PROGRAM Axis05_Rotation_1
VAR
	Axis05: AXIS_REF;											//회전축
	Axis05_MC_Home: FB_HomeBeforeMoveAX8000;
	Axis05_MC_Power: MC_Power;
	Axis05_Status: MC_ReadStatus;
	Axis05_Position_Read: MC_ReadActualPosition;
	Axis05_Velocity_Read: MC_ReadActualVelocity;
	Axis05_Reset: MC_Reset;										//모터 알람 리셋
	Axis05_Stop: MC_Stop;										//모터 정지
	Axis05_Press_Move: MC_MoveAbsolute;
	Axis05_Home_Pos_Move: MC_MoveAbsolute;
	Axis05_Wait_Pos_Move: MC_MoveAbsolute;
	Axis05_Target_Pos_Move: MC_MoveAbsolute;
	Axis05_Work_End_Move: MC_MoveAbsolute;
	Axis05_Jog: MC_Jog;
	
	Always_ON	:	BOOL	:=TRUE	;//상시 ON
	Always_OFF	:	BOOL	:=FALSE	;//상시 OFF

	Home_Interlock			:	BOOL	;
	Home_Pos_Interlock		: 	BOOL	;
	Wait_Pos_Interlock		:	BOOL	;
	Target_Pos_Interlock	:	BOOL	;
	Work_End_POs_Interlock	:	BOOL	;
	Axis05_Calibration: MC_MoveAbsolute;
END_VAR
VAR // added by the converter: edge detectors and wires of the graphical bodies
    _rt1, _rt2, _rt3, _rt4, _rt5, _rt6 : R_TRIG;
    _w1, _w2 : BOOL;
END_VAR

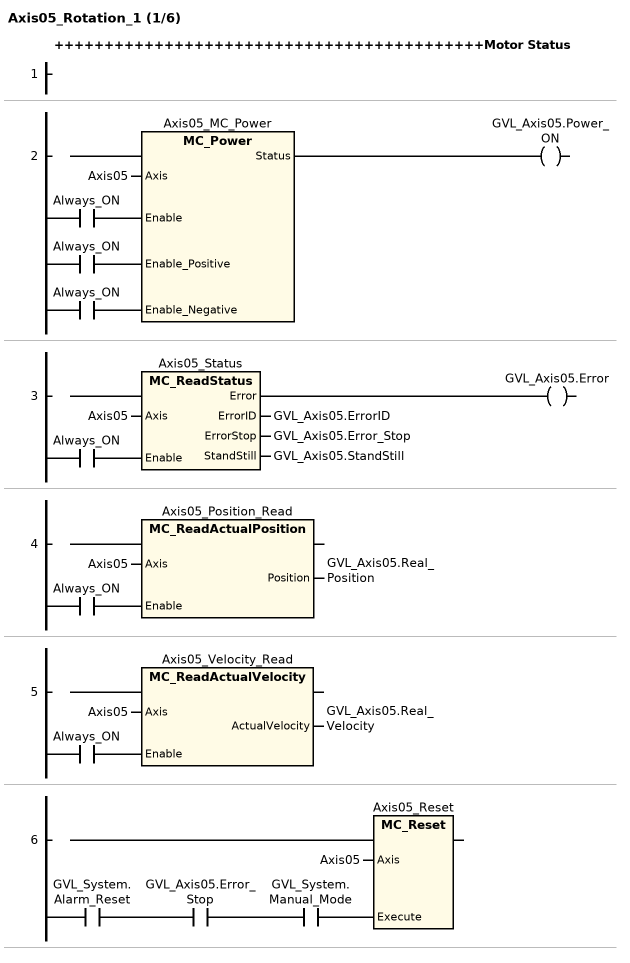
// NETWORK 1: +++++++++++++++++++++++++++++++++++++++++++Motor Status

// NETWORK 2
Axis05_MC_Power(
    Axis := Axis05,
    Enable := Always_ON,
    Enable_Positive := Always_ON,
    Enable_Negative := Always_ON); // MC_Power
GVL_Axis05.Power_ON := Axis05_MC_Power.Status;

// NETWORK 3
Axis05_Status(
    Axis := Axis05,
    Enable := Always_ON,
    Error => GVL_Axis05.Error,
    ErrorID => GVL_Axis05.ErrorID,
    ErrorStop => GVL_Axis05.Error_Stop,
    StandStill => GVL_Axis05.StandStill); // MC_ReadStatus

// NETWORK 4
Axis05_Position_Read(Axis := Axis05, Enable := Always_ON, Position => GVL_Axis05.Real_Position); // MC_ReadActualPosition

// NETWORK 5
Axis05_Velocity_Read(Axis := Axis05, Enable := Always_ON, ActualVelocity => GVL_Axis05.Real_Velocity); // MC_ReadActualVelocity

// NETWORK 6
Axis05_Reset(Axis := Axis05, Execute := GVL_System.Alarm_Reset AND GVL_Axis05.Error_Stop AND GVL_System.Manual_Mode); // MC_Reset

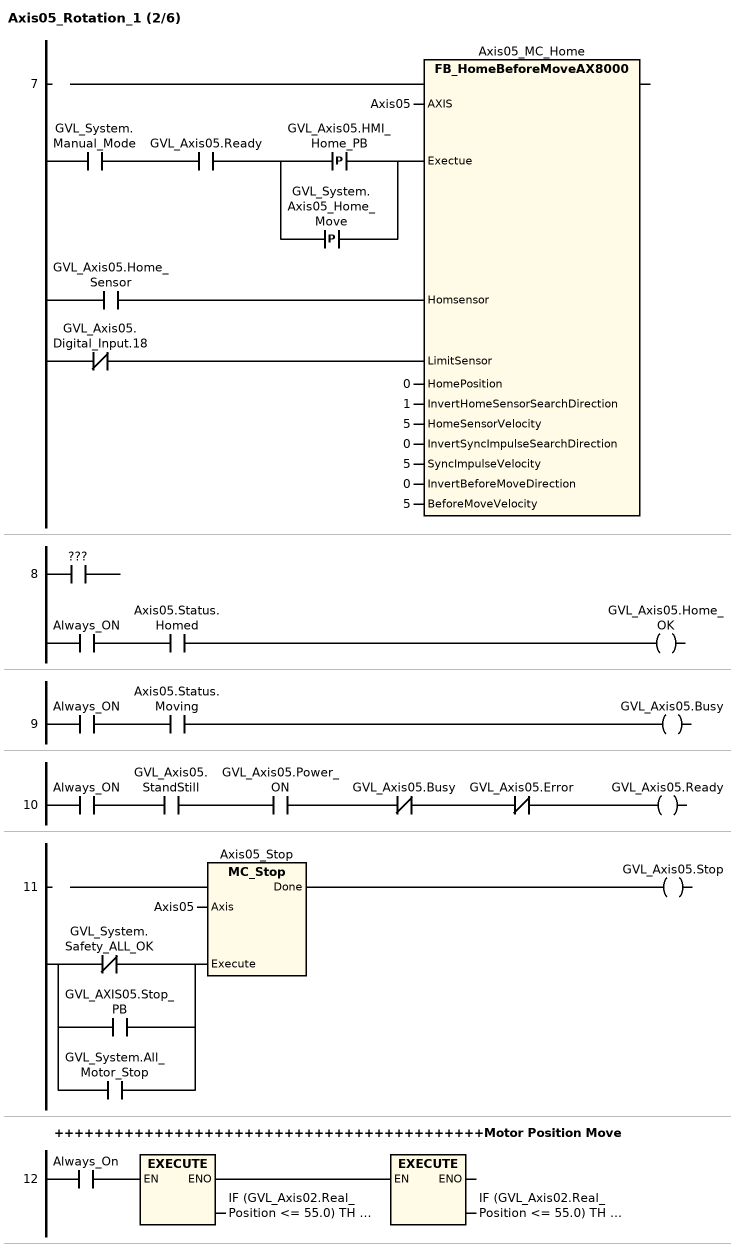
// NETWORK 7
_rt1(CLK := GVL_Axis05.HMI_Home_PB);
_rt2(CLK := GVL_System.Axis05_Home_Move);
Axis05_MC_Home(
    AXIS := Axis05,
    Exectue := GVL_System.Manual_Mode AND GVL_Axis05.Ready AND (_rt1.Q OR _rt2.Q),
    Homsensor := GVL_Axis05.Home_Sensor,
    LimitSensor := NOT GVL_Axis05.Digital_Input.18,
    HomePosition := 0,
    InvertHomeSensorSearchDirection := 1,
    HomeSensorVelocity := 5,
    InvertSyncImpulseSearchDirection := 0,
    SyncImpulseVelocity := 5,
    InvertBeforeMoveDirection := 0,
    BeforeMoveVelocity := 5); // FB_HomeBeforeMoveAX8000

// NETWORK 8
GVL_Axis05.Home_OK := Always_ON AND Axis05.Status.Homed;

// NETWORK 9
GVL_Axis05.Busy := Always_ON AND Axis05.Status.Moving;

// NETWORK 10
GVL_Axis05.Ready := Always_ON AND GVL_Axis05.StandStill AND GVL_Axis05.Power_ON AND NOT GVL_Axis05.Busy AND NOT GVL_Axis05.Error;

// NETWORK 11
Axis05_Stop(Axis := Axis05, Execute := NOT GVL_System.Safety_ALL_OK OR GVL_AXIS05.Stop_PB OR GVL_System.All_Motor_Stop); // MC_Stop
GVL_Axis05.Stop := Axis05_Stop.Done;

// NETWORK 12: +++++++++++++++++++++++++++++++++++++++++++Motor Position Move
_w1 := Always_On;
IF _w1 THEN
    IF (GVL_Axis02.Real_Position <= 55.0) THEN
        Home_Pos_Interlock := TRUE;
    ELSE
        IF (GVL_Axis05.Home_Position_Data >= -1.5) AND 
           (GVL_Axis05.Home_Position_Data <= 2.5) THEN
            Home_Pos_Interlock := TRUE;
        ELSE 
           Home_Pos_Interlock := FALSE;
        END_IF;
    END_IF;
END_IF
IF _w1 THEN
    IF (GVL_Axis02.Real_Position <= 55.0) THEN
        Wait_Pos_Interlock := TRUE;
    ELSE
        IF (GVL_Axis05.Wait_Position_Data >= -1.5) AND 
           (GVL_Axis05.Wait_Position_Data <= 2.5) THEN
            Wait_Pos_Interlock := TRUE;
        ELSE 
           Wait_Pos_Interlock := FALSE;
        END_IF;
    END_IF;
END_IF

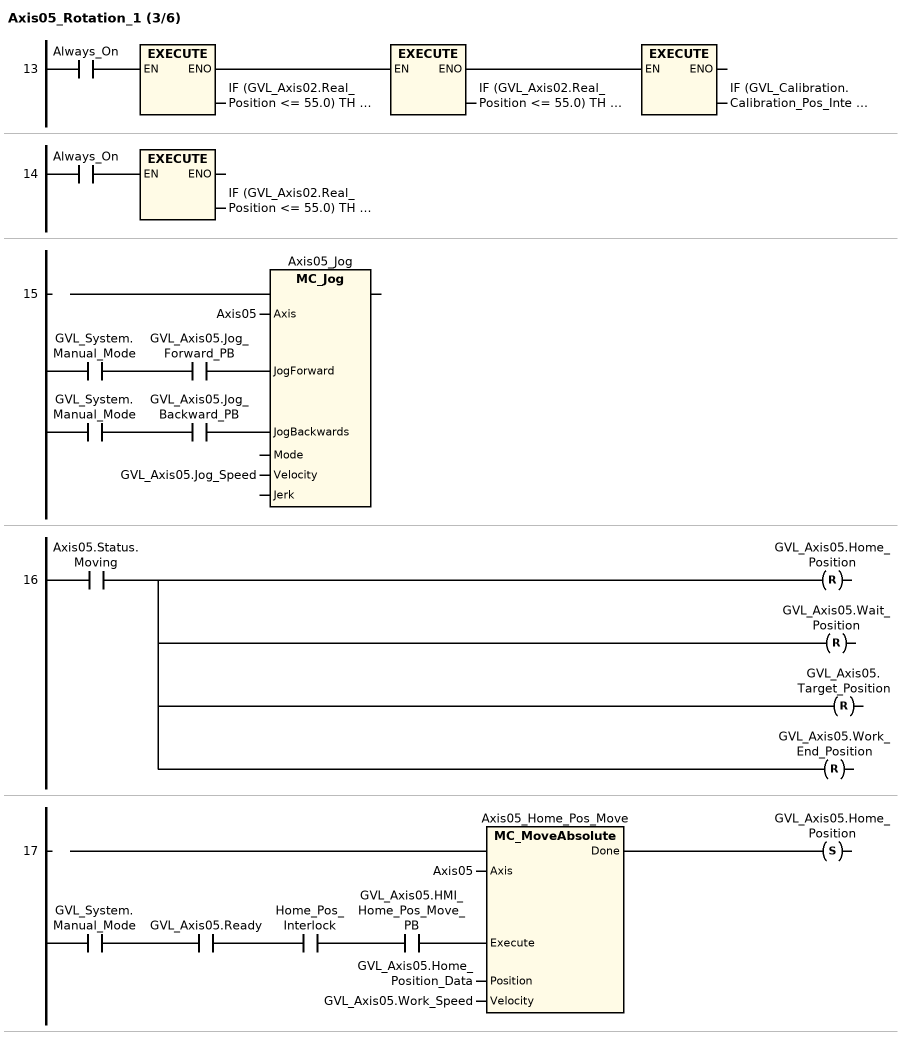
// NETWORK 13
_w2 := Always_On;
IF _w2 THEN
    IF (GVL_Axis02.Real_Position <= 55.0) THEN
        Target_Pos_Interlock := TRUE;
    ELSE
        IF (GVL_Axis05.Target_Position_Data >= -1.5) AND 
           (GVL_Axis05.Target_Position_Data <= 2.5) THEN
            Target_Pos_Interlock := TRUE;
        ELSE 
           Target_Pos_Interlock := FALSE;
        END_IF;
    END_IF;
END_IF
IF _w2 THEN
    IF (GVL_Axis02.Real_Position <= 55.0) THEN
        Work_End_Pos_Interlock := TRUE;
    ELSE
        IF (GVL_Axis05.Work_End_Position_Data >= -1.5) AND 
           (GVL_Axis05.Work_End_Position_Data <= 2.5) THEN
            Work_End_Pos_Interlock := TRUE;
        ELSE 
           Work_End_Pos_Interlock := FALSE;
        END_IF;
    END_IF;
END_IF
IF _w2 THEN
    IF (GVL_Calibration.Calibration_Pos_Interlock = TRUE) AND (Home_Pos_Interlock = TRUE)
    AND (Wait_Pos_Interlock = TRUE) AND (Target_Pos_Interlock = TRUE) AND (Work_End_POs_Interlock = TRUE) THEN
    	GVL_Axis05.Interlock := TRUE;
    	ELSE
    	GVL_Axis05.Interlock := FALSE;	
    
    END_IF
END_IF

// NETWORK 14
IF Always_On THEN
    IF (GVL_Axis02.Real_Position <= 55.0) THEN
        Home_Interlock := TRUE;
    ELSE
           Home_Interlock := FALSE;
    END_IF;
END_IF

// NETWORK 15
Axis05_Jog(
    Axis := Axis05,
    JogForward := GVL_System.Manual_Mode AND GVL_Axis05.Jog_Forward_PB,
    JogBackwards := GVL_System.Manual_Mode AND GVL_Axis05.Jog_Backward_PB,
    Velocity := GVL_Axis05.Jog_Speed); // MC_Jog

// NETWORK 16
GVL_Axis05.Home_Position R= Axis05.Status.Moving;
GVL_Axis05.Wait_Position R= Axis05.Status.Moving;
GVL_Axis05.Target_Position R= Axis05.Status.Moving;
GVL_Axis05.Work_End_Position R= Axis05.Status.Moving;

// NETWORK 17
Axis05_Home_Pos_Move(
    Axis := Axis05,
    Execute := GVL_System.Manual_Mode AND GVL_Axis05.Ready AND Home_Pos_Interlock AND GVL_Axis05.HMI_Home_Pos_Move_PB,
    Position := GVL_Axis05.Home_Position_Data,
    Velocity := GVL_Axis05.Work_Speed); // MC_MoveAbsolute
GVL_Axis05.Home_Position S= Axis05_Home_Pos_Move.Done;

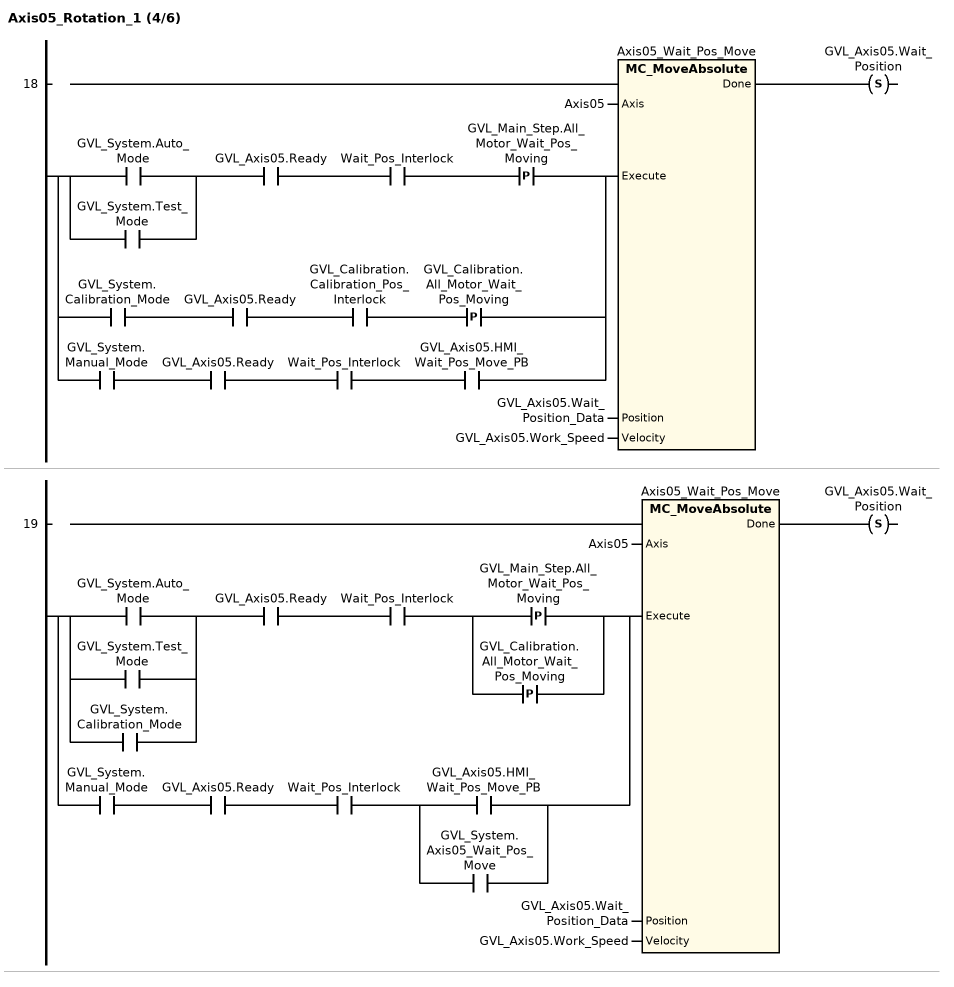
// NETWORK 18
_rt3(CLK := GVL_Main_Step.All_Motor_Wait_Pos_Moving);
_rt4(CLK := GVL_Calibration.All_Motor_Wait_Pos_Moving);
Axis05_Wait_Pos_Move(
    Axis := Axis05,
    Execute := (GVL_System.Auto_Mode OR GVL_System.Test_Mode) AND GVL_Axis05.Ready AND Wait_Pos_Interlock AND _rt3.Q OR GVL_System.Calibration_Mode AND GVL_Axis05.Ready AND GVL_Calibration.Calibration_Pos_Interlock AND _rt4.Q OR GVL_System.Manual_Mode AND GVL_Axis05.Ready AND Wait_Pos_Interlock AND GVL_Axis05.HMI_Wait_Pos_Move_PB,
    Position := GVL_Axis05.Wait_Position_Data,
    Velocity := GVL_Axis05.Work_Speed); // MC_MoveAbsolute
GVL_Axis05.Wait_Position S= Axis05_Wait_Pos_Move.Done;

// NETWORK 19
_rt5(CLK := GVL_Main_Step.All_Motor_Wait_Pos_Moving);
_rt6(CLK := GVL_Calibration.All_Motor_Wait_Pos_Moving);
Axis05_Wait_Pos_Move(
    Axis := Axis05,
    Execute := (GVL_System.Auto_Mode OR GVL_System.Test_Mode OR GVL_System.Calibration_Mode) AND GVL_Axis05.Ready AND Wait_Pos_Interlock AND (_rt5.Q OR _rt6.Q) OR GVL_System.Manual_Mode AND GVL_Axis05.Ready AND Wait_Pos_Interlock AND (GVL_Axis05.HMI_Wait_Pos_Move_PB OR GVL_System.Axis05_Wait_Pos_Move),
    Position := GVL_Axis05.Wait_Position_Data,
    Velocity := GVL_Axis05.Work_Speed); // MC_MoveAbsolute
GVL_Axis05.Wait_Position S= Axis05_Wait_Pos_Move.Done;

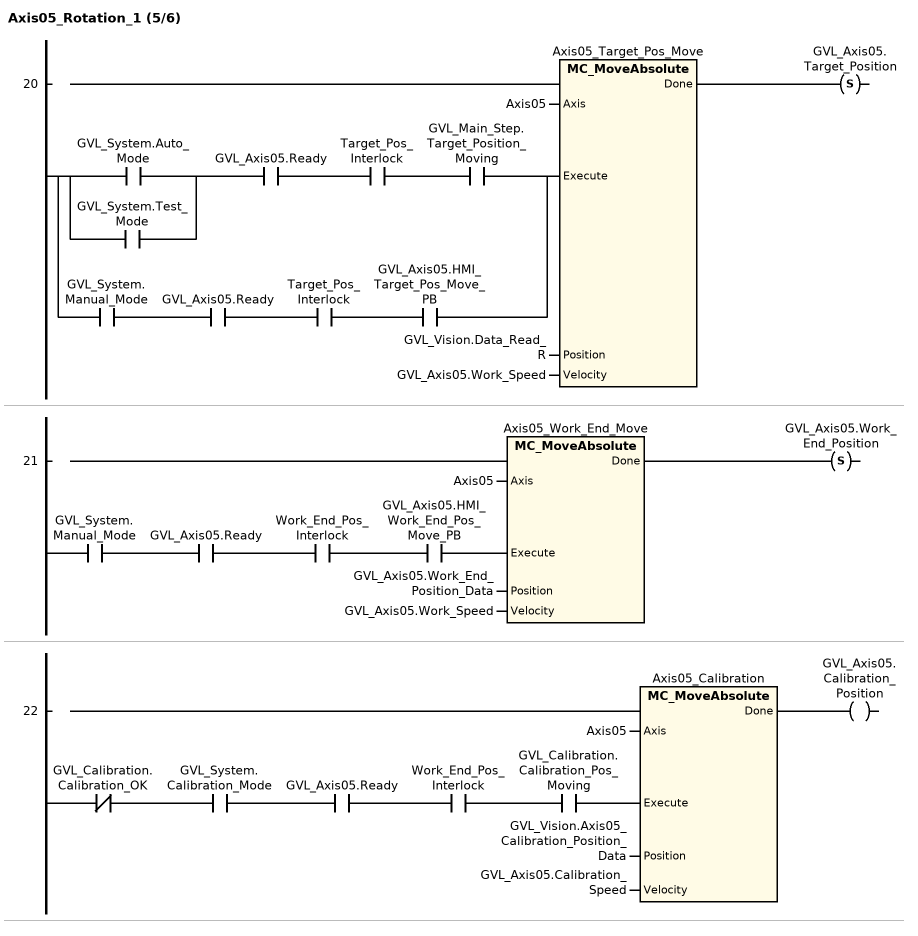
// NETWORK 20
Axis05_Target_Pos_Move(
    Axis := Axis05,
    Execute := (GVL_System.Auto_Mode OR GVL_System.Test_Mode) AND GVL_Axis05.Ready AND Target_Pos_Interlock AND GVL_Main_Step.Target_Position_Moving OR GVL_System.Manual_Mode AND GVL_Axis05.Ready AND Target_Pos_Interlock AND GVL_Axis05.HMI_Target_Pos_Move_PB,
    Position := GVL_Vision.Data_Read_R,
    Velocity := GVL_Axis05.Work_Speed); // MC_MoveAbsolute
GVL_Axis05.Target_Position S= Axis05_Target_Pos_Move.Done;

// NETWORK 21
Axis05_Work_End_Move(
    Axis := Axis05,
    Execute := GVL_System.Manual_Mode AND GVL_Axis05.Ready AND Work_End_Pos_Interlock AND GVL_Axis05.HMI_Work_End_Pos_Move_PB,
    Position := GVL_Axis05.Work_End_Position_Data,
    Velocity := GVL_Axis05.Work_Speed); // MC_MoveAbsolute
GVL_Axis05.Work_End_Position S= Axis05_Work_End_Move.Done;

// NETWORK 22
Axis05_Calibration(
    Axis := Axis05,
    Execute := NOT GVL_Calibration.Calibration_OK AND GVL_System.Calibration_Mode AND GVL_Axis05.Ready AND Work_End_Pos_Interlock AND GVL_Calibration.Calibration_Pos_Moving,
    Position := GVL_Vision.Axis05_Calibration_Position_Data,
    Velocity := GVL_Axis05.Calibration_Speed); // MC_MoveAbsolute
GVL_Axis05.Calibration_Position := Axis05_Calibration.Done;

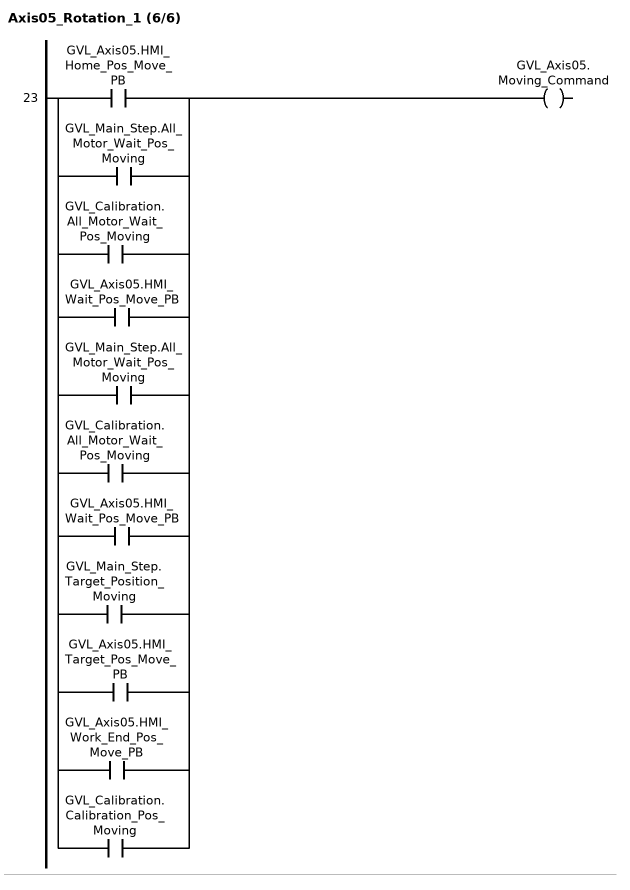
// NETWORK 23
GVL_Axis05.Moving_Command := GVL_Axis05.HMI_Home_Pos_Move_PB OR GVL_Main_Step.All_Motor_Wait_Pos_Moving OR GVL_Calibration.All_Motor_Wait_Pos_Moving OR GVL_Axis05.HMI_Wait_Pos_Move_PB OR GVL_Main_Step.All_Motor_Wait_Pos_Moving OR GVL_Calibration.All_Motor_Wait_Pos_Moving OR GVL_Axis05.HMI_Wait_Pos_Move_PB OR GVL_Main_Step.Target_Position_Moving OR GVL_Axis05.HMI_Target_Pos_Move_PB OR GVL_Axis05.HMI_Work_End_Pos_Move_PB OR GVL_Calibration.Calibration_Pos_Moving;

END_PROGRAM

(* stored: Version 1.1.0.1, ProductVersion 3.1.4024.15
   POU Axis05_Rotation_1: Id {8ca4276f-6e7e-424e-83d3-8273b20242dd}, SpecialFunc None *)
